CIRC {X -222.560,Y -5.949,Z -64.500,A 0.015,B 0.000,C 180.000},{X -221.200,Y -7.047,Z -64.500,A 0.015,B 0.000,C -180.000} C_DIS
LIN {X -189.934,Y -7.047,Z -64.500,A 0.015,B -0.000,C -180.000} C_DIS
CIRC {X -187.101,Y -7.905,Z -64.500,A 0.015,B 0.000,C -180.000},{X -185.219,Y -10.191,Z -64.500,A 0.015,B -0.000,C 180.000} C_DIS
CIRC {X -183.337,Y -12.476,Z -64.500,A 0.015,B 0.000,C -180.000},{X -180.504,Y -13.334,Z -64.500,A 0.015,B 0.000,C 180.000} C_DIS
LIN {X -143.066,Y -13.334,Z -64.500,A 0.015,B 0.000,C -180.000} C_DIS
CIRC {X -141.706,Y -12.236,Z -64.500,A 0.015,B 0.000,C 180.000},{X -142.494,Y -10.675,Z -64.500,A 0.015,B 0.000,C 180.000} C_DIS
LIN {X -188.981,Y 10.128,Z -64.500,A 0.015,B 0.000,C -180.000} C_DIS
CIRC {X -190.225,Y 10.769,Z -64.500,A 0.015,B -0.000,C -180.000},{X -191.395,Y 11.536,Z -64.500,A 0.015,B 0.000,C 180.000} C_DIS
CIRC {X -192.522,Y 12.363,Z -64.500,A 0.015,B 0.000,C -180.000},{X -193.645,Y 13.193,Z -64.500,A 0.015,B 0.000,C 180.000} C_DIS
CIRC {X -196.671,Y 14.214,Z -64.500,A 0.015,B 0.000,C 180.000},{X -199.722,Y 13.270,Z -64.500,A 0.015,B 0.000,C 180.000} C_DIS
CIRC {X -200.946,Y 12.397,Z -64.500,A 0.015,B -0.000,C -180.000},{X -202.158,Y 11.509,Z -64.500,A 0.015,B -0.000,C 180.000} C_DIS
CIRC {X -203.413,Y 10.678,Z -64.500,A 0.015,B -0.000,C -180.000},{X -204.749,Y 9.986,Z -64.500,A 0.015,B 0.000,C -180.000} C_DIS
LIN {X -250.991,Y -10.675,Z -64.500,A 0.015,B 0.000,C 180.000} C_DIS
CIRC {X -251.778,Y -12.236,Z -64.500,A 0.015,B -0.000,C 180.000},{X -250.418,Y -13.334,Z -64.500,A 0.015,B 0.000,C 180.000} C_DIS
LIN {X -180.504,Y -13.334,Z -64.500,A 0.015,B 0.000,C 180.000} C_DIS
CIRC {X -177.670,Y -14.192,Z -64.500,A 0.015,B 0.000,C 180.000},{X -175.788,Y -16.478,Z -64.500,A 0.015,B 0.000,C 180.000} C_DIS
CIRC {X -173.906,Y -18.764,Z -64.500,A 0.015,B -0.000,C 180.000},{X -171.073,Y -19.622,Z -64.500,A 0.015,B 0.000,C -180.000} C_DIS
LIN {X -113.868,Y -19.622,Z -64.500,A 0.015,B 0.000,C -180.000} C_DIS
CIRC {X -112.507,Y -18.523,Z -64.500,A 0.015,B -0.000,C -180.000},{X -113.295,Y -16.962,Z -64.500,A 0.015,B 0.000,C 180.000} C_DIS
LIN {X -186.463,Y 15.702,Z -64.500,A 0.015,B 0.000,C 180.000} C_DIS
CIRC {X -188.899,Y 17.071,Z -64.500,A 0.015,B 0.000,C -180.000},{X -191.059,Y 18.844,Z -64.500,A 0.015,B 0.000,C -180.000} C_DIS
CIRC {X -192.975,Y 20.865,Z -64.500,A 0.015,B 0.000,C -180.000},{X -194.736,Y 23.023,Z -64.500,A 0.015,B -0.000,C 180.000} C_DIS
CIRC {X -196.819,Y 24.036,Z -64.500,A 0.015,B -0.000,C 180.000},{X -198.863,Y 22.946,Z -64.500,A 0.015,B -0.000,C 180.000} C_DIS
CIRC {X -199.831,Y 21.635,Z -64.500,A 0.015,B -0.000,C 180.000},{X -200.867,Y 20.377,Z -64.500,A 0.015,B 0.000,C 180.000} C_DIS
CIRC {X -202.011,Y 19.212,Z -64.500,A 0.015,B 0.000,C -180.000},{X -203.291,Y 18.199,Z -64.500,A 0.015,B -0.000,C -180.000} C_DIS
CIRC {X -204.263,Y 17.507,Z -64.500,A 0.015,B 0.000,C 180.000},{X -205.219,Y 16.793,Z -64.500,A 0.015,B 0.000,C 180.000} C_DIS
CIRC {X -206.209,Y 16.122,Z -64.500,A 0.015,B 0.000,C 180.000},{X -207.269,Y 15.569,Z -64.500,A 0.015,B 0.000,C 180.000} C_DIS
LIN {X -280.209,Y -16.962,Z -64.500,A 0.015,B 0.000,C 180.000} C_DIS
CIRC {X -280.996,Y -18.523,Z -64.500,A 0.015,B 0.000,C 180.000},{X -279.636,Y -19.622,Z -64.500,A 0.015,B 0.000,C -180.000} C_DIS
LIN {X -171.073,Y -19.622,Z -64.500,A 0.015,B 0.000,C -180.000} C_DIS
LIN {X -170.464,Y -19.466,Z -64.330,A 0.015,B 0.000,C -180.000} C_DIS
LIN {X -170.105,Y -19.174,Z -63.865,A 0.015,B -0.000,C 180.000} C_DIS
LIN {X -170.004,Y -19.038,Z -63.230,A 0.015,B 0.000,C 180.000} C_DIS
$VEL.CP = 1.00000
LIN {X -170.004,Y -19.038,Z 11.000,A 0.015,B 0.000,C 180.000} C_DIS
$VEL.CP = 1.00000
LIN {X -328.228,Y 254.055,Z 11.000,A 0.015,B 0.000,C -180.000} C_DIS
$VEL.CP = 1.00000
LIN {X -328.228,Y 254.055,Z -42.731,A 0.015,B -0.000,C -180.000} C_DIS
$VEL.CP = 0.10000
LIN {X -328.066,Y 254.037,Z -43.353,A 0.015,B 0.000,C -180.000} C_DIS
LIN {X -327.621,Y 254.009,Z -43.816,A 0.015,B 0.000,C -180.000} C_DIS
LIN {X -327.005,Y 254.024,Z -44.000,A 0.015,B 0.000,C -180.000} C_DIS
LIN {X -321.768,Y 258.048,Z -44.244,A 0.015,B 0.000,C 180.000} C_DIS
LIN {X -323.357,Y 264.459,Z -44.488,A 0.015,B 0.000,C -180.000} C_DIS
LIN {X -329.867,Y 265.572,Z -44.732,A 0.015,B 0.000,C 180.000} C_DIS
LIN {X -333.495,Y 260.054,Z -44.976,A 0.015,B 0.000,C -180.000} C_DIS
LIN {X -329.894,Y 254.518,Z -45.220,A 0.015,B -0.000,C -180.000} C_DIS
LIN {X -323.379,Y 255.600,Z -45.464,A 0.015,B -0.000,C 180.000} C_DIS
LIN {X -321.759,Y 262.002,Z -45.708,A 0.015,B 0.000,C 180.000} C_DIS
LIN {X -326.976,Y 266.052,Z -45.952,A 0.015,B 0.000,C 180.000} C_DIS
LIN {X -332.777,Y 262.895,Z -46.196,A 0.015,B 0.000,C -180.000} C_DIS
LIN {X -332.209,Y 256.315,Z -46.440,A 0.015,B -0.000,C 180.000} C_DIS
LIN {X -325.953,Y 254.199,Z -46.685,A 0.015,B 0.000,C 180.000} C_DIS
LIN {X -321.507,Y 259.082,Z -46.929,A 0.015,B 0.000,C 180.000} C_DIS
LIN {X -324.200,Y 265.113,Z -47.173,A 0.015,B 0.000,C 180.000} C_DIS
LIN {X -330.804,Y 265.062,Z -47.417,A 0.015,B 0.000,C -180.000} C_DIS
LIN {X -333.404,Y 258.991,Z -47.661,A 0.015,B 0.000,C 180.000} C_DIS
LIN {X -328.883,Y 254.176,Z -47.905,A 0.015,B 0.000,C -180.000} C_DIS
LIN {X -322.660,Y 256.388,Z -48.149,A 0.015,B 0.000,C 180.000} C_DIS
LIN {X -322.194,Y 262.976,Z -48.393,A 0.015,B 0.000,C -180.000} C_DIS
LIN {X -328.042,Y 266.044,Z -48.637,A 0.015,B 0.000,C -180.000} C_DIS
LIN {X -333.196,Y 261.914,Z -48.881,A 0.015,B -0.000,C -180.000} C_DIS
LIN {X -331.479,Y 255.537,Z -49.125,A 0.015,B 0.000,C 180.000} C_DIS
LIN {X -324.948,Y 254.556,Z -49.369,A 0.015,B -0.000,C 180.000} C_DIS
LIN {X -321.431,Y 260.146,Z -49.613,A 0.015,B 0.000,C 180.000} C_DIS
LIN {X -325.144,Y 265.608,Z -49.857,A 0.015,B 0.000,C -180.000} C_DIS
LIN {X -331.636,Y 264.395,Z -50.101,A 0.015,B 0.000,C 180.000} C_DIS
LIN {X -333.126,Y 257.961,Z -50.345,A 0.015,B 0.000,C 180.000} C_DIS
LIN {X -327.828,Y 254.018,Z -50.589,A 0.015,B 0.000,C 180.000} C_DIS
LIN {X -322.092,Y 257.291,Z -50.833,A 0.015,B -0.000,C 180.000} C_DIS
LIN {X -322.793,Y 263.858,Z -51.077,A 0.015,B 0.000,C 180.000} C_DIS
LIN {X -329.091,Y 265.848,Z -51.321,A 0.015,B 0.000,C 180.000} C_DIS
LIN {X -333.437,Y 260.875,Z -51.565,A 0.015,B 0.000,C -180.000} C_DIS
LIN {X -330.623,Y 254.900,Z -51.810,A 0.015,B -0.000,C 180.000} C_DIS
LIN {X -324.021,Y 255.085,Z -52.054,A 0.015,B 0.000,C -180.000} C_DIS
LIN {X -321.544,Y 261.207,Z -52.298,A 0.015,B 0.000,C -180.000} C_DIS
LIN {X -326.161,Y 265.929,Z -52.542,A 0.015,B 0.000,C 180.000} C_DIS
LIN {X -332.338,Y 263.592,Z -52.786,A 0.015,B 0.000,C -180.000} C_DIS
LIN {X -332.672,Y 256.996,Z -53.030,A 0.015,B 0.000,C 180.000} C_DIS
LIN {X -326.762,Y 254.047,Z -53.274,A 0.015,B 0.000,C -180.000} C_DIS
LIN {X -321.692,Y 258.280,Z -53.518,A 0.015,B 0.000,C -180.000} C_DIS
LIN {X -323.539,Y 264.621,Z -53.762,A 0.015,B 0.000,C -180.000} C_DIS
LIN {X -330.088,Y 265.470,Z -54.006,A 0.015,B 0.000,C 180.000} C_DIS
LIN {X -333.491,Y 259.810,Z -54.250,A 0.015,B -0.000,C -180.000} C_DIS
LIN {X -329.668,Y 254.424,Z -54.494,A 0.015,B 0.000,C -180.000} C_DIS
LIN {X -323.202,Y 255.768,Z -54.738,A 0.015,B 0.000,C 180.000} C_DIS
LIN {X -321.843,Y 262.231,Z -54.982,A 0.015,B 0.000,C 180.000} C_DIS
LIN {X -327.219,Y 266.067,Z -55.226,A 0.015,B -0.000,C -180.000} C_DIS
LIN {X -332.888,Y 262.678,Z -55.470,A 0.015,B 0.000,C -180.000} C_DIS
LIN {X -332.054,Y 256.126,Z -55.714,A 0.015,B 0.000,C 180.000} C_DIS
LIN {X -325.718,Y 254.264,Z -55.958,A 0.015,B 0.000,C 180.000} C_DIS
LIN {X -321.473,Y 259.324,Z -56.202,A 0.015,B -0.000,C 180.000} C_DIS
LIN {X -324.407,Y 265.240,Z -56.446,A 0.015,B 0.000,C -180.000} C_DIS
LIN {X -331.004,Y 264.923,Z -56.690,A 0.015,B 0.000,C 180.000} C_DIS
LIN {X -333.356,Y 258.752,Z -56.935,A 0.015,B 0.000,C 180.000} C_DIS
LIN {X -328.645,Y 254.123,Z -57.179,A 0.015,B 0.000,C 180.000} C_DIS
LIN {X -322.517,Y 256.585,Z -57.423,A 0.015,B 0.000,C 180.000} C_DIS
LIN {X -322.317,Y 263.187,Z -57.667,A 0.015,B -0.000,C 180.000} C_DIS
LIN {X -328.285,Y 266.015,Z -57.911,A 0.015,B 0.000,C 180.000} C_DIS
LIN {X -333.268,Y 261.681,Z -58.155,A 0.015,B 0.000,C 180.000} C_DIS
LIN {X -331.293,Y 255.379,Z -58.399,A 0.015,B -0.000,C 180.000} C_DIS
LIN {X -324.728,Y 254.662,Z -58.643,A 0.015,B 0.000,C -180.000} C_DIS
LIN {X -321.441,Y 260.390,Z -58.887,A 0.015,B 0.000,C 180.000} C_DIS
LIN {X -325.371,Y 265.697,Z -59.131,A 0.015,B 0.000,C -180.000} C_DIS
LIN {X -331.809,Y 264.223,Z -59.375,A 0.015,B 0.000,C -180.000} C_DIS
LIN {X -333.037,Y 257.734,Z -59.619,A 0.015,B 0.000,C -180.000} C_DIS
LIN {X -327.585,Y 254.008,Z -59.863,A 0.015,B -0.000,C -180.000} C_DIS
LIN {X -321.986,Y 257.511,Z -60.107,A 0.015,B -0.000,C 180.000} C_DIS
LIN {X -322.951,Y 264.044,Z -60.351,A 0.015,B 0.000,C 180.000} C_DIS
LIN {X -329.324,Y 265.777,Z -60.595,A 0.015,B 0.000,C -180.000} C_DIS
LIN {X -333.466,Y 260.633,Z -60.839,A 0.015,B -0.000,C -180.000} C_DIS
LIN {X -330.413,Y 254.777,Z -61.083,A 0.015,B 0.000,C 180.000} C_DIS
LIN {X -323.824,Y 255.228,Z -61.327,A 0.015,B 0.000,C 180.000} C_DIS
LIN {X -321.597,Y 261.445,Z -61.571,A 0.015,B 0.000,C 180.000} C_DIS
LIN {X -326.400,Y 265.977,Z -61.815,A 0.015,B 0.000,C -180.000} C_DIS
LIN {X -332.478,Y 263.392,Z -62.060,A 0.015,B 0.000,C 180.000} C_DIS
LIN {X -332.544,Y 256.788,Z -62.304,A 0.015,B 0.000,C -180.000} C_DIS
LIN {X -326.520,Y 254.081,Z -62.548,A 0.015,B 0.000,C -180.000} C_DIS
LIN {X -321.626,Y 258.515,Z -62.792,A 0.015,B 0.000,C 180.000} C_DIS
LIN {X -323.727,Y 264.776,Z -63.036,A 0.015,B 0.000,C 180.000} C_DIS
LIN {X -330.306,Y 265.360,Z -63.280,A 0.015,B 0.000,C 180.000} C_DIS
LIN {X -333.477,Y 259.566,Z -63.524,A 0.015,B 0.000,C 180.000} C_DIS
LIN {X -329.440,Y 254.340,Z -63.768,A 0.015,B 0.000,C -180.000} C_DIS
LIN {X -323.033,Y 255.944,Z -64.012,A 0.015,B 0.000,C -180.000} C_DIS
LIN {X -321.936,Y 262.456,Z -64.256,A 0.015,B 0.000,C -180.000} C_DIS
LIN {X -327.463,Y 266.072,Z -64.500,A 0.015,B 0.000,C -180.000} C_DIS
LIN {X -327.817,Y 266.072,Z -64.500,A 0.015,B 0.000,C 180.000} C_DIS
CIRC {X -329.824,Y 265.240,Z -64.500,A 0.015,B -0.000,C 180.000},{X -330.656,Y 263.233,Z -64.500,A 0.015,B -0.000,C 180.000} C_DIS
LIN {X -330.655,Y 221.906,Z -64.500,A 0.015,B 0.000,C 180.000} C_DIS
CIRC {X -329.566,Y 220.761,Z -64.500,A 0.015,B 0.000,C -180.000},{X -328.368,Y 221.792,Z -64.500,A 0.015,B -0.000,C 180.000} C_DIS
LIN {X -324.247,Y 262.950,Z -64.500,A 0.015,B 0.000,C 180.000} C_DIS
CIRC {X -324.967,Y 265.138,Z -64.500,A 0.015,B 0.000,C 180.000},{X -327.071,Y 266.072,Z -64.500,A 0.015,B 0.000,C 180.000} C_DIS
LIN {X -327.463,Y 266.072,Z -64.500,A 0.015,B 0.000,C -180.000} C_DIS
CIRC {X -329.644,Y 266.865,Z -64.500,A 0.015,B 0.000,C 180.000},{X -330.806,Y 268.874,Z -64.500,A 0.015,B 0.000,C -180.000} C_DIS
CIRC {X -332.544,Y 270.781,Z -64.500,A 0.015,B 0.000,C 180.000},{X -335.012,Y 270.031,Z -64.500,A 0.015,B 0.000,C 180.000} C_DIS
CIRC {X -335.708,Y 268.856,Z -64.500,A 0.015,B -0.000,C 180.000},{X -335.950,Y 267.512,Z -64.500,A 0.015,B 0.000,C 180.000} C_DIS
LIN {X -335.947,Y 181.701,Z -64.500,A 0.015,B 0.000,C -180.000} C_DIS
CIRC {X -334.834,Y 179.879,Z -64.500,A 0.015,B 0.000,C -180.000},{X -332.704,Y 180.038,Z -64.500,A 0.015,B 0.000,C 180.000} C_DIS
LIN {X -328.199,Y 183.276,Z -64.500,A 0.015,B 0.000,C 180.000} C_DIS
CIRC {X -327.124,Y 184.463,Z -64.500,A 0.015,B 0.000,C 180.000},{X -326.633,Y 185.987,Z -64.500,A 0.015,B 0.000,C 180.000} C_DIS
LIN {X -318.461,Y 267.601,Z -64.500,A 0.015,B -0.000,C 180.000} C_DIS
CIRC {X -319.329,Y 270.239,Z -64.500,A 0.015,B -0.000,C 180.000},{X -321.867,Y 271.365,Z -64.500,A 0.015,B 0.000,C 180.000} C_DIS
LIN {X -332.097,Y 271.365,Z -64.500,A 0.015,B 0.000,C -180.000} C_DIS
CIRC {X -333.700,Y 271.016,Z -64.500,A 0.015,B 0.000,C 180.000},{X -335.012,Y 270.031,Z -64.500,A 0.015,B 0.000,C -180.000} C_DIS
CIRC {X -337.395,Y 267.835,Z -64.500,A 0.015,B -0.000,C 180.000},{X -340.211,Y 266.233,Z -64.500,A 0.015,B -0.000,C -180.000} C_DIS
CIRC {X -342.792,Y 264.080,Z -64.500,A 0.015,B 0.000,C -180.000},{X -343.759,Y 260.861,Z -64.500,A 0.015,B 0.000,C -180.000} C_DIS
LIN {X -343.757,Y 166.471,Z -64.500,A 0.015,B 0.000,C -180.000} C_DIS
CIRC {X -342.643,Y 164.649,Z -64.500,A 0.015,B -0.000,C 180.000},{X -340.514,Y 164.808,Z -64.500,A 0.015,B 0.000,C -180.000} C_DIS
LIN {X -323.839,Y 176.792,Z -64.500,A 0.015,B 0.000,C 180.000} C_DIS
CIRC {X -320.407,Y 180.584,Z -64.500,A 0.015,B -0.000,C 180.000},{X -318.838,Y 185.452,Z -64.500,A 0.015,B 0.000,C -180.000} C_DIS
LIN {X -309.830,Y 275.411,Z -64.500,A 0.015,B -0.000,C -180.000} C_DIS
CIRC {X -310.698,Y 278.049,Z -64.500,A 0.015,B 0.000,C -180.000},{X -313.236,Y 279.175,Z -64.500,A 0.015,B 0.000,C -180.000} C_DIS

; Continue running program as cascaded execution
Machining3()

END
